ABB RobotStudio station: 6700_EGM_20220705-170627.rsstn

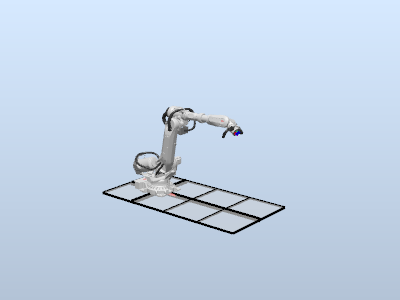
Station Station (saved by RobotStudio 22.2.9947.0)
Controller IRB6700_140_285_MH6
  mechanical unit ROB_1: IRB6700_140_285_MH6_04, 6 joints, base frame (0, 0, 0) mm
Layout (positions relative to the parent item):
  - IRB6700_140_285_MH6_04 [mechanism, from Robots\IRB6700_140_285_MH6_04.rslib] at (0, 0, 0) mm; joint values [0, 0.3155, -0.334, -0.3936, 0.5236, 0.3757] (rad or m)
